
FUNCTION CB_abs_sint : INT


TITLE = ' Absolute value of a number '
VERSION : '1.0'
AUTHOR  : CB
NAME    : abs_int
FAMILY  : TNI

VAR_INPUT
    IN : INT;
END_VAR

VAR_TEMP

END_VAR

BEGIN

CB_abs_sint := ABS(IN);

END_FUNCTION
